(* IEC 61131-3 sources: Piper/src/Ar/Piper, 3 files *)

(* ---- Piper.typ ---- *)
(*
* File: Piper.typ
* Copyright (c) 2023 Loupe
* https://loupe.team
*
* This file is part of the Piper Library, licensed under the MIT License.
*)

TYPE
	Piper_typ : 	STRUCT
		IN : Piper_IN_typ;
		OUT : Piper_OUT_typ;
		Internal : Piper_Internal_typ;
		IO : Piper_IO_typ;
	END_STRUCT;
	Piper_IN_typ : 	STRUCT
		CMD : Piper_IN_CMD_typ;
		CFG : Piper_IN_CFG_typ;
	END_STRUCT;
	Piper_IN_CFG_typ : 	STRUCT
		BootCycles : UINT := PIPER_DEFAULT_BOOTING_CYCLES;
		LoggerName : STRING[LOG_STRLEN_LOGGERNAME];
	END_STRUCT;
	Piper_IN_CMD_typ : 	STRUCT
		Reset : BOOL;
		Start : BOOL;
		Stop : BOOL;
		Hold : BOOL;
		Unhold : BOOL;
		Suspend : BOOL;
		Unsuspend : BOOL;
		Abort : BOOL;
		Clear : BOOL;
		BypassAll : BOOL;
		AcknowledgeError : BOOL;
	END_STRUCT;
	Piper_IO_typ : 	STRUCT
		iMainInterface : Module_Interface_typ;
		oMainInterface : Module_Interface_typ;
	END_STRUCT;
	Piper_OUT_typ : 	STRUCT
		Error : UINT;
		ErrorString : STRING[80];
		State : MACH_ST_enum; (*The current PackML state of system*)
		SubState : DINT; (*The current step within the PackML state*)
		BusyModule : UDINT; (*The first module that is busy*)
		ErrorModule : UDINT; (*The first module that has an error*)
		SubStateRequestModule : UDINT; (*The module that requested the next step*)
	END_STRUCT;
	Piper_Internal_typ : 	STRUCT
		NextSubState : DINT; (*The next step that should be executed when the current step is complete*)
		ResponseStatus : PIPER_RESPONSE_ST; (*The state of the response of the current step*)
		ModuleList : ARRAY[0..MAI_PIPER_MODULES]OF UDINT; (*The pipes that are attached to this manager*)
		ModuleNames : ARRAY[0..MAI_PIPER_MODULES]OF STRING[80]; (*Names of the modules to ensure uniqueness after download*)
		NumberModules : DINT;
		BootCycles : UINT;
	END_STRUCT;
	Module_Interface_typ : 	STRUCT
		ModuleName : STRING[80];
		ModuleStatus : STRING[80];
		PiperState : MACH_ST_enum;
		PiperSubState : DINT;
		ModuleResponse : MACH_ST_enum;
		ModuleSubStateRequest : DINT;
		ModuleCommand : Piper_IN_CMD_typ;
		ModuleBypass : BOOL;
		ModuleIsBypassed : BOOL;
	END_STRUCT;
	Piper_Module_Internal_typ : 	STRUCT
		Added : BOOL;
		ModuleIndex : UDINT;
	END_STRUCT;
	PIPER_RESPONSE_ST :
		(
		PIPER_RESPONSE_ST_NONE,
		PIPER_RESPONSE_ST_ERROR,
		PIPER_RESPONSE_ST_STEP_DONE,
		PIPER_RESPONSE_ST_NEXT_STEP,
		PIPER_RESPONSE_ST_STATE_DONE,
		PIPER_RESPONSE_ST_BUSY
		);
	MACH_ST_enum :
		(
		MACH_ST_NOT_READY := 0, (*0*)
		MACH_ST_BOOTING := 1, (*1*)
		MACH_ST_BOOTED,
		MACH_ST_ERROR,
		MACH_ST_CLEARING,
		MACH_ST_STOPPED, (*5*)
		MACH_ST_STARTING,
		MACH_ST_IDLE,
		MACH_ST_SUSPENDED,
		MACH_ST_EXECUTE,
		MACH_ST_STOPPING, (*10*)
		MACH_ST_ABORTING,
		MACH_ST_ABORTED,
		MACH_ST_HOLDING,
		MACH_ST_HELD,
		MACH_ST_UNHOLDING, (*15*)
		MACH_ST_SUSPENDING,
		MACH_ST_UNSUSPENDING,
		MACH_ST_RESETTING,
		MACH_ST_COMPLETING,
		MACH_ST_COMPLETE, (*20*)
		MACH_ST_BYPASSED,
		MACH_ST_ (*22*)
		);
END_TYPE

(* ---- Piper.fun ---- *)
(*
* File: Piper.fun
* Copyright (c) 2023 Loupe
* https://loupe.team
*
* This file is part of the Piper Library, licensed under the MIT License.
*)

FUNCTION Piper_fn_Cyclic : BOOL (*Master Cyclic function*) (*$GROUP=User*)
	VAR_INPUT
		Piper : Piper_typ;
	END_VAR
END_FUNCTION

FUNCTION Piper_Remote_fn_Cyclic : BOOL (*Master Cyclic function*) (*$GROUP=User*)
	VAR_INPUT
		Piper : Piper_typ;
		IsRemote : BOOL;
	END_VAR
END_FUNCTION

FUNCTION_BLOCK Piper_Module_Fub (*Implements the interface to a pipe*) (*$GROUP=User*)
	VAR_INPUT
		Piper : REFERENCE TO Piper_typ;
		ModuleInterface : REFERENCE TO Module_Interface_typ;
	END_VAR
	VAR
		internal : Piper_Module_Internal_typ;
	END_VAR
END_FUNCTION_BLOCK
(*
Internal Piper Functions
*)

FUNCTION Piper_changeState : BOOL (*Performs and logs a state change*) (*$GROUP=User*)
	VAR_INPUT
		Piper : Piper_typ;
		State : MACH_ST_enum;
	END_VAR
END_FUNCTION

FUNCTION Piper_checkResponses : BOOL (*Reads the status of Pipes*) (*$GROUP=User*)
	VAR_INPUT
		Piper : Piper_typ;
	END_VAR
END_FUNCTION

FUNCTION Piper_getState_remote : BOOL (*Gets state and substate from main Piper*) (*$GROUP=User*)
	VAR_INPUT
		Piper : Piper_typ;
	END_VAR
END_FUNCTION

FUNCTION Piper_handleResponseState : BOOL (*This function looks at the response state and decides what Step or State to enter next*) (*$GROUP=User*)
	VAR_INPUT
		Piper : Piper_typ;
	END_VAR
END_FUNCTION

FUNCTION Piper_PackML : BOOL (*Implements PackML state machine for Piper*) (*$GROUP=User*)
	VAR_INPUT
		Piper : Piper_typ;
	END_VAR
END_FUNCTION

FUNCTION Piper_setCommand : BOOL (*Sets commands to the subsystems*) (*$GROUP=User*)
	VAR_INPUT
		Piper : Piper_typ;
	END_VAR
END_FUNCTION

FUNCTION Piper_setSubstate : BOOL (*Sets the substate given the current internal response status*) (*$GROUP=User*)
	VAR_INPUT
		Piper : Piper_typ;
	END_VAR
END_FUNCTION

(*
Internal Helper Functions
*)

FUNCTION PackMLStateString : BOOL (*Returns a string for the given PackML state*) (*$GROUP=User*)
	VAR_INPUT
		State : MACH_ST_enum;
		String : STRING[80];
	END_VAR
END_FUNCTION

FUNCTION PiperModuleDoneWithState : BOOL (*Returns whether the given module is done with its current state*)
	VAR_INPUT
		ModuleInterface : Module_Interface_typ;
	END_VAR
END_FUNCTION

FUNCTION PiperModuleDoneWithSubstate : BOOL (*Returns whether the given module is done with its current substate*)
	VAR_INPUT
		ModuleInterface : Module_Interface_typ;
	END_VAR
END_FUNCTION

FUNCTION Piper_getBusyModules : UINT (*This function finds modules reporting busy to Piper*)
	VAR_INPUT
		Piper : Piper_typ;
		pModuleArray : UDINT;
		numModules : UINT;
		offset : UINT;
	END_VAR
END_FUNCTION

(* ---- Piper.var ---- *)
(*
* File: Piper.var
* Copyright (c) 2023 Loupe
* https://loupe.team
*
* This file is part of the Piper Library, licensed under the MIT License.
*)

VAR CONSTANT
	PIPER_DEFAULT_BOOTING_CYCLES : UINT := 50;
	MAI_PIPER_MODULES : USINT := 99;
	PIPER_DEFAULT_LOGGERNAME : STRING[LOG_STRLEN_LOGGERNAME] := 'App';
	IDLE_SUBSTATE : DINT := 65535;
END_VAR
